# B&R Automation Studio project Teknologia25
Automation Studio 6.3.4.31; technology packages: mapp6D 3.4.1, mappView 6.3.2, OpcUaCs 6.0.0

## Configuration Config1

CPU X20EM0613, AutomationRuntime 6.0.2, Build 11.3.0, Vc 6.0.0

### Task classes (Cpu.sw)
```
Cyclic#1 (cycle 2000 us, tolerance 0 us):
  Main <- Main.Main.prg
  Acp6D <- Acp6D.Acp6D.prg
Cyclic#8:
  Robot <- Robot.Robot.prg
NcDataObjects: McDriveLog
Binaries: udbdef, mvLoader, mvConfig, OpcUaSrv, TCData, FWRules, ArSvcReg, BRRole, asfw, Role, ashwac, UaCsConfig, sysconf, iomap, Config_2, Config, Config_1, ashwd, User, arconfig
Libraries: operator, runtime, astime, AsIecCon, standard, RandLib, AsBrStr, AsBrMath, FileIO, BrAbbRws, AsHttp, ArEventLog, ArSsl, Crypto, AsIODiag, brdkMU, AsSem, sys_lib, brsystem, brdkSTR, MTFilter, MTTypes, MTLinAlg, AsUDP, AsTCP, comUtil, strUtil, McAcp6D, McBase, MpBase, brfiDemo
```

### Hardware
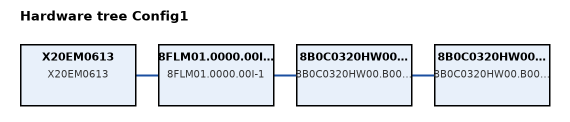
```
8B0C0320HW00.B00-1 : 8B0C0320HW00.B00-1 v1.0.1.3 (NodeNumber=3)  [PLK1 -> 8FLM01.0000.00I-1.PLK2 [Cable Type=PowerlinkCable, Length=10, Version=1.0.0.3]; PLK2 -> 8B0C0320HW00.B00-1_a.PLK1 [Cable Type=PowerlinkCable, Length=10, Version=1.0.0.3]]
  FunctionModel = DirectControl
  Supervision = off
  OutputVoltage = 58000
  CurrentLimitation = Used
  OutputCurrentLimit = 20000
  OutputCurrentLimitTime = 20
  ConfigOutputState = on
8B0C0320HW00.B00-1_a : 8B0C0320HW00.B00-1 v1.0.1.3  [PLK1 -> 8B0C0320HW00.B00-1.PLK2 [Cable Type=PowerlinkCable, Length=10, Version=1.0.0.3]]
  FunctionModel = DirectControl
  Supervision = off
  OutputVoltage = 58000
  CurrentLimitation = Used
  OutputCurrentLimit = 20000
  OutputCurrentLimitTime = 20
  ConfigOutputState = on
8FLM01.0000.00I-1 : 8FLM01.0000.00I-1 v1.0.0.1 (NodeNumber=239)  [PLK1 -> X20EM0613.IF3 [Cable Type=PowerlinkCable, Length=10, Version=1.0.0.3]; PLK2 -> 8B0C0320HW00.B00-1.PLK1 [Cable Type=PowerlinkCable, Length=10, Version=1.0.0.3]]
  Supervision = off
X20EM0613 : X20EM0613 v1.1.1.0
  Connector IF2:
    ActivateDevice = 1
    Mode = Manual
    InternetAddress = 192.168.125.201
    SubnetMask = 255.255.255.0
    ActivateSnmp = 2
  ConfigurationID = Teknologia25_Config1
  TimerDeviceType = EPLX2X
  TimerDevice = X20EM0613.IF3
  TaskClassIdleTime = 2000
  Cyclic1Duration = 2000
  Cyclic1Tolerance = 0
  FileDevice1
  FileDeviceName1 = 6DData
  FileDevicePath1 = USER_PATH
  ActivateFtpServer = 1
  FTPProtocol = 1
  FtpUser1
  FtpUsername1 = br
  FtpUserPassword1 = LZr6u6a2FqeMuMrXqkQdYPSQXL3utztiI9HOjYTJN4M=  // admin
  FtpUserSalt1 = xnOKDKah
  FTPAccessRight1 = 0
  FTPdevice1 = ALL
  ActivateWebServer = 1
  WebServerProtocol = 1
  WebServerPort = 8087
  ActivateSdm = 1
```

### IoMap.iom - X20EM0613/IoMap.iom
```iecst
VAR_CONFIG
	 Cyclic#1.::gCommInput.Array[0] AT %IW."8FLM01.0000.00I-1".EPL_FB_IN_0_I2007_S01;
	 Cyclic#1.::gCommInput.Array[1] AT %IW."8FLM01.0000.00I-1".EPL_FB_IN_1_I2007_S02;
	 Cyclic#1.::gCommInput.Array[2] AT %IW."8FLM01.0000.00I-1".EPL_FB_IN_2_I2007_S03;
	 Cyclic#1.::gCommInput.Array[3] AT %IW."8FLM01.0000.00I-1".EPL_FB_IN_3_I2007_S04;
	 Cyclic#1.::gCommInput.Array[4] AT %IW."8FLM01.0000.00I-1".EPL_FB_IN_4_I2007_S05;
	 Cyclic#1.::gCommInput.Array[5] AT %IW."8FLM01.0000.00I-1".EPL_FB_IN_5_I2007_S06;
	 Cyclic#1.::gCommInput.Array[6] AT %IW."8FLM01.0000.00I-1".EPL_FB_IN_6_I2007_S07;
	 Cyclic#1.::gCommInput.Array[7] AT %IW."8FLM01.0000.00I-1".EPL_FB_IN_7_I2007_S08;
	 Cyclic#1.::gCommInput.Array[8] AT %IW."8FLM01.0000.00I-1".EPL_FB_IN_8_I2007_S09;
	 Cyclic#1.::gCommInput.Array[9] AT %IW."8FLM01.0000.00I-1".EPL_FB_IN_9_I2007_S0A;
	 Cyclic#1.::gCommInput.Array[10] AT %IW."8FLM01.0000.00I-1".EPL_FB_IN_10_I2007_S0B;
	 Cyclic#1.::gCommInput.Array[11] AT %IW."8FLM01.0000.00I-1".EPL_FB_IN_11_I2007_S0C;
	 Cyclic#1.::gCommInput.Array[12] AT %IW."8FLM01.0000.00I-1".EPL_FB_IN_12_I2007_S0D;
	 Cyclic#1.::gCommInput.Array[13] AT %IW."8FLM01.0000.00I-1".EPL_FB_IN_13_I2007_S0E;
	 Cyclic#1.::gCommInput.Array[14] AT %IW."8FLM01.0000.00I-1".EPL_FB_IN_14_I2007_S0F;
	 Cyclic#1.::gCommInput.Array[15] AT %IW."8FLM01.0000.00I-1".EPL_FB_IN_15_I2007_S10;
	 Cyclic#1.::gCommInput.Array[16] AT %IW."8FLM01.0000.00I-1".EPL_FB_IN_16_I2007_S11;
	 Cyclic#1.::gCommInput.Array[17] AT %IW."8FLM01.0000.00I-1".EPL_FB_IN_17_I2007_S12;
	 Cyclic#1.::gCommInput.Array[18] AT %IW."8FLM01.0000.00I-1".EPL_FB_IN_18_I2007_S13;
	 Cyclic#1.::gCommInput.Array[19] AT %IW."8FLM01.0000.00I-1".EPL_FB_IN_19_I2007_S14;
	 Cyclic#1.::gCommInput.Array[20] AT %IW."8FLM01.0000.00I-1".EPL_FB_IN_20_I2007_S15;
	 Cyclic#1.::gCommInput.Array[21] AT %IW."8FLM01.0000.00I-1".EPL_FB_IN_21_I2007_S16;
	 Cyclic#1.::gCommInput.Array[22] AT %IW."8FLM01.0000.00I-1".EPL_FB_IN_22_I2007_S17;
	 Cyclic#1.::gCommInput.Array[23] AT %IW."8FLM01.0000.00I-1".EPL_FB_IN_23_I2007_S18;
	 Cyclic#1.::gCommInput.Array[24] AT %IW."8FLM01.0000.00I-1".EPL_FB_IN_24_I2007_S19;
	 Cyclic#1.::gCommInput.Array[25] AT %IW."8FLM01.0000.00I-1".EPL_FB_IN_25_I2007_S1A;
	 Cyclic#1.::gCommInput.Array[26] AT %IW."8FLM01.0000.00I-1".EPL_FB_IN_26_I2007_S1B;
	 Cyclic#1.::gCommInput.Array[27] AT %IW."8FLM01.0000.00I-1".EPL_FB_IN_27_I2007_S1C;
	 Cyclic#1.::gCommInput.Array[28] AT %IW."8FLM01.0000.00I-1".EPL_FB_IN_28_I2007_S1D;
	 Cyclic#1.::gCommInput.Array[29] AT %IW."8FLM01.0000.00I-1".EPL_FB_IN_29_I2007_S1E;
	 Cyclic#1.::gCommInput.Array[30] AT %IW."8FLM01.0000.00I-1".EPL_FB_IN_30_I2007_S1F;
	 Cyclic#1.::gCommInput.Array[31] AT %IW."8FLM01.0000.00I-1".EPL_FB_IN_31_I2007_S20;
	 Cyclic#1.::gCommInput.Array[32] AT %IW."8FLM01.0000.00I-1".EPL_FB_IN_32_I2007_S21;
	 Cyclic#1.::gCommInput.Array[33] AT %IW."8FLM01.0000.00I-1".EPL_FB_IN_33_I2007_S22;
	 Cyclic#1.::gCommInput.Array[34] AT %IW."8FLM01.0000.00I-1".EPL_FB_IN_34_I2007_S23;
	 Cyclic#1.::gCommInput.Array[35] AT %IW."8FLM01.0000.00I-1".EPL_FB_IN_35_I2007_S24;
	 Cyclic#1.::gCommInput.Array[36] AT %IW."8FLM01.0000.00I-1".EPL_FB_IN_36_I2007_S25;
	 Cyclic#1.::gCommInput.Array[37] AT %IW."8FLM01.0000.00I-1".EPL_FB_IN_37_I2007_S26;
	 Cyclic#1.::gCommInput.Array[38] AT %IW."8FLM01.0000.00I-1".EPL_FB_IN_38_I2007_S27;
	 Cyclic#1.::gCommInput.Array[39] AT %IW."8FLM01.0000.00I-1".EPL_FB_IN_39_I2007_S28;
	 Cyclic#1.::gCommInput.Array[40] AT %IW."8FLM01.0000.00I-1".EPL_FB_IN_40_I2007_S29;
	 Cyclic#1.::gCommInput.Array[41] AT %IW."8FLM01.0000.00I-1".EPL_FB_IN_41_I2007_S2A;
	 Cyclic#1.::gCommInput.Array[42] AT %IW."8FLM01.0000.00I-1".EPL_FB_IN_42_I2007_S2B;
	 Cyclic#1.::gCommInput.Array[43] AT %IW."8FLM01.0000.00I-1".EPL_FB_IN_43_I2007_S2C;
	 Cyclic#1.::gCommInput.Array[44] AT %IW."8FLM01.0000.00I-1".EPL_FB_IN_44_I2007_S2D;
	 Cyclic#1.::gCommInput.Array[45] AT %IW."8FLM01.0000.00I-1".EPL_FB_IN_45_I2007_S2E;
	 Cyclic#1.::gCommInput.Array[46] AT %IW."8FLM01.0000.00I-1".EPL_FB_IN_46_I2007_S2F;
	 Cyclic#1.::gCommInput.Array[47] AT %IW."8FLM01.0000.00I-1".EPL_FB_IN_47_I2007_S30;
	 Cyclic#1.::gCommInput.Array[48] AT %IW."8FLM01.0000.00I-1".EPL_FB_IN_48_I2007_S31;
	 Cyclic#1.::gCommInput.Array[49] AT %IW."8FLM01.0000.00I-1".EPL_FB_IN_49_I2007_S32;
	 Cyclic#1.::gCommInput.Array[50] AT %IW."8FLM01.0000.00I-1".EPL_FB_IN_50_I2007_S33;
	 Cyclic#1.::gCommInput.Array[51] AT %IW."8FLM01.0000.00I-1".EPL_FB_IN_51_I2007_S34;
	 Cyclic#1.::gCommInput.Array[52] AT %IW."8FLM01.0000.00I-1".EPL_FB_IN_52_I2007_S35;
	 Cyclic#1.::gCommInput.Array[53] AT %IW."8FLM01.0000.00I-1".EPL_FB_IN_53_I2007_S36;
	 Cyclic#1.::gCommInput.Array[54] AT %IW."8FLM01.0000.00I-1".EPL_FB_IN_54_I2007_S37;
	 Cyclic#1.::gCommInput.Array[55] AT %IW."8FLM01.0000.00I-1".EPL_FB_IN_55_I2007_S38;
	 Cyclic#1.::gCommInput.Array[56] AT %IW."8FLM01.0000.00I-1".EPL_FB_IN_56_I2007_S39;
	 Cyclic#1.::gCommInput.Array[57] AT %IW."8FLM01.0000.00I-1".EPL_FB_IN_57_I2007_S3A;
	 Cyclic#1.::gCommInput.Array[58] AT %IW."8FLM01.0000.00I-1".EPL_FB_IN_58_I2007_S3B;
	 Cyclic#1.::gCommInput.Array[59] AT %IW."8FLM01.0000.00I-1".EPL_FB_IN_59_I2007_S3C;
	 Cyclic#1.::gCommInput.Array[60] AT %IW."8FLM01.0000.00I-1".EPL_FB_IN_60_I2007_S3D;
	 Cyclic#1.::gCommInput.Array[61] AT %IW."8FLM01.0000.00I-1".EPL_FB_IN_61_I2007_S3E;
	 Cyclic#1.::gCommInput.Array[62] AT %IW."8FLM01.0000.00I-1".EPL_FB_IN_62_I2007_S3F;
	 Cyclic#1.::gCommInput.Array[63] AT %IW."8FLM01.0000.00I-1".EPL_FB_IN_63_I2007_S40;
	 Cyclic#1.::gCommInput.Array[64] AT %IW."8FLM01.0000.00I-1".EPL_FB_IN_64_I2007_S41;
	 Cyclic#1.::gCommInput.Array[65] AT %IW."8FLM01.0000.00I-1".EPL_FB_IN_65_I2007_S42;
	 Cyclic#1.::gCommInput.Array[66] AT %IW."8FLM01.0000.00I-1".EPL_FB_IN_66_I2007_S43;
	 Cyclic#1.::gCommInput.Array[67] AT %IW."8FLM01.0000.00I-1".EPL_FB_IN_67_I2007_S44;
	 Cyclic#1.::gCommInput.Array[68] AT %IW."8FLM01.0000.00I-1".EPL_FB_IN_68_I2007_S45;
	 Cyclic#1.::gCommInput.Array[69] AT %IW."8FLM01.0000.00I-1".EPL_FB_IN_69_I2007_S46;
	 Cyclic#1.::gCommInput.Array[70] AT %IW."8FLM01.0000.00I-1".EPL_FB_IN_70_I2007_S47;
	 Cyclic#1.::gCommInput.Array[71] AT %IW."8FLM01.0000.00I-1".EPL_FB_IN_71_I2007_S48;
	 Cyclic#1.::gCommInput.Array[72] AT %IW."8FLM01.0000.00I-1".EPL_FB_IN_72_I2007_S49;
	 Cyclic#1.::gCommInput.Array[73] AT %IW."8FLM01.0000.00I-1".EPL_FB_IN_73_I2007_S4A;
	 Cyclic#1.::gCommInput.Array[74] AT %IW."8FLM01.0000.00I-1".EPL_FB_IN_74_I2007_S4B;
	 Cyclic#1.::gCommInput.Array[75] AT %IW."8FLM01.0000.00I-1".EPL_FB_IN_75_I2007_S4C;
	 Cyclic#1.::gCommInput.Array[76] AT %IW."8FLM01.0000.00I-1".EPL_FB_IN_76_I2007_S4D;
	 Cyclic#1.::gCommInput.Array[77] AT %IW."8FLM01.0000.00I-1".EPL_FB_IN_77_I2007_S4E;
	 Cyclic#1.::gCommInput.Array[78] AT %IW."8FLM01.0000.00I-1".EPL_FB_IN_78_I2007_S4F;
	 Cyclic#1.::gCommInput.Array[79] AT %IW."8FLM01.0000.00I-1".EPL_FB_IN_79_I2007_S50;
	 Cyclic#1.::gCommInput.Array[80] AT %IW."8FLM01.0000.00I-1".EPL_FB_IN_80_I2007_S51;
	 Cyclic#1.::gCommInput.Array[81] AT %IW."8FLM01.0000.00I-1".EPL_FB_IN_81_I2007_S52;
	 Cyclic#1.::gCommInput.Array[82] AT %IW."8FLM01.0000.00I-1".EPL_FB_IN_82_I2007_S53;
	 Cyclic#1.::gCommInput.Array[83] AT %IW."8FLM01.0000.00I-1".EPL_FB_IN_83_I2007_S54;
	 Cyclic#1.::gCommInput.Array[84] AT %IW."8FLM01.0000.00I-1".EPL_FB_IN_84_I2007_S55;
	 Cyclic#1.::gCommInput.Array[85] AT %IW."8FLM01.0000.00I-1".EPL_FB_IN_85_I2007_S56;
	 Cyclic#1.::gCommInput.Array[86] AT %IW."8FLM01.0000.00I-1".EPL_FB_IN_86_I2007_S57;
	 Cyclic#1.::gCommInput.Array[87] AT %IW."8FLM01.0000.00I-1".EPL_FB_IN_87_I2007_S58;
	 Cyclic#1.::gCommInput.Array[88] AT %IW."8FLM01.0000.00I-1".EPL_FB_IN_88_I2007_S59;
	 Cyclic#1.::gCommInput.Array[89] AT %IW."8FLM01.0000.00I-1".EPL_FB_IN_89_I2007_S5A;
	 Cyclic#1.::gCommInput.Array[90] AT %IW."8FLM01.0000.00I-1".EPL_FB_IN_90_I2007_S5B;
	 Cyclic#1.::gCommInput.Array[91] AT %IW."8FLM01.0000.00I-1".EPL_FB_IN_91_I2007_S5C;
	 Cyclic#1.::gCommInput.Array[92] AT %IW."8FLM01.0000.00I-1".EPL_FB_IN_92_I2007_S5D;
	 Cyclic#1.::gCommInput.Array[93] AT %IW."8FLM01.0000.00I-1".EPL_FB_IN_93_I2007_S5E;
	 Cyclic#1.::gCommInput.Array[94] AT %IW."8FLM01.0000.00I-1".EPL_FB_IN_94_I2007_S5F;
	 Cyclic#1.::gCommInput.Array[95] AT %IW."8FLM01.0000.00I-1".EPL_FB_IN_95_I2007_S60;
	 Cyclic#1.::gCommInput.Array[96] AT %IW."8FLM01.0000.00I-1".EPL_FB_IN_96_I2007_S61;
	 Cyclic#1.::gCommInput.Array[97] AT %IW."8FLM01.0000.00I-1".EPL_FB_IN_97_I2007_S62;
	 Cyclic#1.::gCommInput.Array[98] AT %IW."8FLM01.0000.00I-1".EPL_FB_IN_98_I2007_S63;
	 Cyclic#1.::gCommInput.Array[99] AT %IW."8FLM01.0000.00I-1".EPL_FB_IN_99_I2007_S64;
	 Cyclic#1.::gCommInput.Array[100] AT %IW."8FLM01.0000.00I-1".EPL_FB_IN_100_I2007_S65;
	 Cyclic#1.::gCommInput.Array[101] AT %IW."8FLM01.0000.00I-1".EPL_FB_IN_101_I2007_S66;
	 Cyclic#1.::gCommInput.Array[102] AT %IW."8FLM01.0000.00I-1".EPL_FB_IN_102_I2007_S67;
	 Cyclic#1.::gCommInput.Array[103] AT %IW."8FLM01.0000.00I-1".EPL_FB_IN_103_I2007_S68;
	 Cyclic#1.::gCommInput.Array[104] AT %IW."8FLM01.0000.00I-1".EPL_FB_IN_104_I2007_S69;
	 Cyclic#1.::gCommInput.Array[105] AT %IW."8FLM01.0000.00I-1".EPL_FB_IN_105_I2007_S6A;
	 Cyclic#1.::gCommInput.Array[106] AT %IW."8FLM01.0000.00I-1".EPL_FB_IN_106_I2007_S6B;
	 Cyclic#1.::gCommInput.Array[107] AT %IW."8FLM01.0000.00I-1".EPL_FB_IN_107_I2007_S6C;
	 Cyclic#1.::gCommInput.Array[108] AT %IW."8FLM01.0000.00I-1".EPL_FB_IN_108_I2007_S6D;
	 Cyclic#1.::gCommInput.Array[109] AT %IW."8FLM01.0000.00I-1".EPL_FB_IN_109_I2007_S6E;
	 Cyclic#1.::gCommInput.Array[110] AT %IW."8FLM01.0000.00I-1".EPL_FB_IN_110_I2007_S6F;
	 Cyclic#1.::gCommInput.Array[111] AT %IW."8FLM01.0000.00I-1".EPL_FB_IN_111_I2007_S70;
	 Cyclic#1.::gCommInput.Array[112] AT %IW."8FLM01.0000.00I-1".EPL_FB_IN_112_I2007_S71;
	 Cyclic#1.::gCommInput.Array[113] AT %IW."8FLM01.0000.00I-1".EPL_FB_IN_113_I2007_S72;
	 Cyclic#1.::gCommInput.Array[114] AT %IW."8FLM01.0000.00I-1".EPL_FB_IN_114_I2007_S73;
	 Cyclic#1.::gCommInput.Array[115] AT %IW."8FLM01.0000.00I-1".EPL_FB_IN_115_I2007_S74;
	 Cyclic#1.::gCommInput.Array[116] AT %IW."8FLM01.0000.00I-1".EPL_FB_IN_116_I2007_S75;
	 Cyclic#1.::gCommInput.Array[117] AT %IW."8FLM01.0000.00I-1".EPL_FB_IN_117_I2007_S76;
	 Cyclic#1.::gCommInput.Array[118] AT %IW."8FLM01.0000.00I-1".EPL_FB_IN_118_I2007_S77;
	 Cyclic#1.::gCommInput.Array[119] AT %IW."8FLM01.0000.00I-1".EPL_FB_IN_119_I2007_S78;
	 Cyclic#1.::gCommInput.Array[120] AT %IW."8FLM01.0000.00I-1".EPL_FB_IN_120_I2007_S79;
	 Cyclic#1.::gCommInput.Array[121] AT %IW."8FLM01.0000.00I-1".EPL_FB_IN_121_I2007_S7A;
	 Cyclic#1.::gCommInput.Array[122] AT %IW."8FLM01.0000.00I-1".EPL_FB_IN_122_I2007_S7B;
	 Cyclic#1.::gCommInput.Array[123] AT %IW."8FLM01.0000.00I-1".EPL_FB_IN_123_I2007_S7C;
	 Cyclic#1.::gCommInput.Array[124] AT %IW."8FLM01.0000.00I-1".EPL_FB_IN_124_I2007_S7D;
	 Cyclic#1.::gCommInput.Array[125] AT %IW."8FLM01.0000.00I-1".EPL_FB_IN_125_I2007_S7E;
	 Cyclic#1.::gCommInput.Array[126] AT %IW."8FLM01.0000.00I-1".EPL_FB_IN_126_I2007_S7F;
	 Cyclic#1.::gCommInput.Array[127] AT %IW."8FLM01.0000.00I-1".EPL_FB_IN_127_I2007_S80;
	 Cyclic#1.::gCommInput.Array[128] AT %IW."8FLM01.0000.00I-1".EPL_FB_IN_128_I2007_S81;
	 Cyclic#1.::gCommInput.Array[129] AT %IW."8FLM01.0000.00I-1".EPL_FB_IN_129_I2007_S82;
	 Cyclic#1.::gCommInput.Array[130] AT %IW."8FLM01.0000.00I-1".EPL_FB_IN_130_I2007_S83;
	 Cyclic#1.::gCommInput.Array[131] AT %IW."8FLM01.0000.00I-1".EPL_FB_IN_131_I2007_S84;
	 Cyclic#1.::gCommInput.Array[132] AT %IW."8FLM01.0000.00I-1".EPL_FB_IN_132_I2007_S85;
	 Cyclic#1.::gCommInput.Array[133] AT %IW."8FLM01.0000.00I-1".EPL_FB_IN_133_I2007_S86;
	 Cyclic#1.::gCommInput.Array[134] AT %IW."8FLM01.0000.00I-1".EPL_FB_IN_134_I2007_S87;
	 Cyclic#1.::gCommInput.Array[135] AT %IW."8FLM01.0000.00I-1".EPL_FB_IN_135_I2007_S88;
	 Cyclic#1.::gCommInput.Array[136] AT %IW."8FLM01.0000.00I-1".EPL_FB_IN_136_I2007_S89;
	 Cyclic#1.::gCommInput.Array[137] AT %IW."8FLM01.0000.00I-1".EPL_FB_IN_137_I2007_S8A;
	 Cyclic#1.::gCommInput.Array[138] AT %IW."8FLM01.0000.00I-1".EPL_FB_IN_138_I2007_S8B;
	 Cyclic#1.::gCommInput.Array[139] AT %IW."8FLM01.0000.00I-1".EPL_FB_IN_139_I2007_S8C;
	 Cyclic#1.::gCommInput.Array[140] AT %IW."8FLM01.0000.00I-1".EPL_FB_IN_140_I2007_S8D;
	 Cyclic#1.::gCommInput.Array[141] AT %IW."8FLM01.0000.00I-1".EPL_FB_IN_141_I2007_S8E;
	 Cyclic#1.::gCommInput.Array[142] AT %IW."8FLM01.0000.00I-1".EPL_FB_IN_142_I2007_S8F;
	 Cyclic#1.::gCommInput.Array[143] AT %IW."8FLM01.0000.00I-1".EPL_FB_IN_143_I2007_S90;
	 Cyclic#1.::gCommInput.Array[144] AT %IW."8FLM01.0000.00I-1".EPL_FB_IN_144_I2007_S91;
	 Cyclic#1.::gCommInput.Array[145] AT %IW."8FLM01.0000.00I-1".EPL_FB_IN_145_I2007_S92;
	 Cyclic#1.::gCommInput.Array[146] AT %IW."8FLM01.0000.00I-1".EPL_FB_IN_146_I2007_S93;
	 Cyclic#1.::gCommInput.Array[147] AT %IW."8FLM01.0000.00I-1".EPL_FB_IN_147_I2007_S94;
	 Cyclic#1.::gCommInput.Array[148] AT %IW."8FLM01.0000.00I-1".EPL_FB_IN_148_I2007_S95;
	 Cyclic#1.::gCommInput.Array[149] AT %IW."8FLM01.0000.00I-1".EPL_FB_IN_149_I2007_S96;
	 Cyclic#1.::gCommInput.Array[150] AT %IW."8FLM01.0000.00I-1".EPL_FB_IN_150_I2007_S97;
	 Cyclic#1.::gCommInput.Array[151] AT %IW."8FLM01.0000.00I-1".EPL_FB_IN_151_I2007_S98;
	 Cyclic#1.::gCommInput.Array[152] AT %IW."8FLM01.0000.00I-1".EPL_FB_IN_152_I2007_S99;
	 Cyclic#1.::gCommInput.Array[153] AT %IW."8FLM01.0000.00I-1".EPL_FB_IN_153_I2007_S9A;
	 Cyclic#1.::gCommInput.Array[154] AT %IW."8FLM01.0000.00I-1".EPL_FB_IN_154_I2007_S9B;
	 Cyclic#1.::gCommInput.Array[155] AT %IW."8FLM01.0000.00I-1".EPL_FB_IN_155_I2007_S9C;
	 Cyclic#1.::gCommInput.Array[156] AT %IW."8FLM01.0000.00I-1".EPL_FB_IN_156_I2007_S9D;
	 Cyclic#1.::gCommInput.Array[157] AT %IW."8FLM01.0000.00I-1".EPL_FB_IN_157_I2007_S9E;
	 Cyclic#1.::gCommInput.Array[158] AT %IW."8FLM01.0000.00I-1".EPL_FB_IN_158_I2007_S9F;
	 Cyclic#1.::gCommInput.Array[159] AT %IW."8FLM01.0000.00I-1".EPL_FB_IN_159_I2007_SA0;
	 Cyclic#1.::gCommInput.Array[160] AT %IW."8FLM01.0000.00I-1".EPL_FB_IN_160_I2007_SA1;
	 Cyclic#1.::gCommInput.Array[161] AT %IW."8FLM01.0000.00I-1".EPL_FB_IN_161_I2007_SA2;
	 Cyclic#1.::gCommInput.Array[162] AT %IW."8FLM01.0000.00I-1".EPL_FB_IN_162_I2007_SA3;
	 Cyclic#1.::gCommInput.Array[163] AT %IW."8FLM01.0000.00I-1".EPL_FB_IN_163_I2007_SA4;
	 Cyclic#1.::gCommInput.Array[164] AT %IW."8FLM01.0000.00I-1".EPL_FB_IN_164_I2007_SA5;
	 Cyclic#1.::gCommInput.Array[165] AT %IW."8FLM01.0000.00I-1".EPL_FB_IN_165_I2007_SA6;
	 Cyclic#1.::gCommInput.Array[166] AT %IW."8FLM01.0000.00I-1".EPL_FB_IN_166_I2007_SA7;
	 Cyclic#1.::gCommInput.Array[167] AT %IW."8FLM01.0000.00I-1".EPL_FB_IN_167_I2007_SA8;
	 Cyclic#1.::gCommInput.Array[168] AT %IW."8FLM01.0000.00I-1".EPL_FB_IN_168_I2007_SA9;
	 Cyclic#1.::gCommInput.Array[169] AT %IW."8FLM01.0000.00I-1".EPL_FB_IN_169_I2007_SAA;
	 Cyclic#1.::gCommInput.Array[170] AT %IW."8FLM01.0000.00I-1".EPL_FB_IN_170_I2007_SAB;
	 Cyclic#1.::gCommInput.Array[171] AT %IW."8FLM01.0000.00I-1".EPL_FB_IN_171_I2007_SAC;
	 Cyclic#1.::gCommInput.Array[172] AT %IW."8FLM01.0000.00I-1".EPL_FB_IN_172_I2007_SAD;
	 Cyclic#1.::gCommInput.Array[173] AT %IW."8FLM01.0000.00I-1".EPL_FB_IN_173_I2007_SAE;
	 Cyclic#1.::gCommInput.Array[174] AT %IW."8FLM01.0000.00I-1".EPL_FB_IN_174_I2007_SAF;
	 Cyclic#1.::gCommInput.Array[175] AT %IW."8FLM01.0000.00I-1".EPL_FB_IN_175_I2007_SB0;
	 Cyclic#1.::gCommInput.Array[176] AT %IW."8FLM01.0000.00I-1".EPL_FB_IN_176_I2007_SB1;
	 Cyclic#1.::gCommInput.Array[177] AT %IW."8FLM01.0000.00I-1".EPL_FB_IN_177_I2007_SB2;
	 Cyclic#1.::gCommInput.Array[178] AT %IW."8FLM01.0000.00I-1".EPL_FB_IN_178_I2007_SB3;
	 Cyclic#1.::gCommInput.Array[179] AT %IW."8FLM01.0000.00I-1".EPL_FB_IN_179_I2007_SB4;
	 Cyclic#1.::gCommInput.Array[180] AT %IW."8FLM01.0000.00I-1".EPL_FB_IN_180_I2007_SB5;
	 Cyclic#1.::gCommInput.Array[181] AT %IW."8FLM01.0000.00I-1".EPL_FB_IN_181_I2007_SB6;
	 Cyclic#1.::gCommInput.Array[182] AT %IW."8FLM01.0000.00I-1".EPL_FB_IN_182_I2007_SB7;
	 Cyclic#1.::gCommInput.Array[183] AT %IW."8FLM01.0000.00I-1".EPL_FB_IN_183_I2007_SB8;
	 Cyclic#1.::gCommInput.Array[184] AT %IW."8FLM01.0000.00I-1".EPL_FB_IN_184_I2007_SB9;
	 Cyclic#1.::gCommInput.Array[185] AT %IW."8FLM01.0000.00I-1".EPL_FB_IN_185_I2007_SBA;
	 Cyclic#1.::gCommInput.Array[186] AT %IW."8FLM01.0000.00I-1".EPL_FB_IN_186_I2007_SBB;
	 Cyclic#1.::gCommInput.Array[187] AT %IW."8FLM01.0000.00I-1".EPL_FB_IN_187_I2007_SBC;
	 Cyclic#1.::gCommInput.Array[188] AT %IW."8FLM01.0000.00I-1".EPL_FB_IN_188_I2007_SBD;
	 Cyclic#1.::gCommInput.Array[189] AT %IW."8FLM01.0000.00I-1".EPL_FB_IN_189_I2007_SBE;
	 Cyclic#1.::gCommInput.Array[190] AT %IW."8FLM01.0000.00I-1".EPL_FB_IN_190_I2007_SBF;
	 Cyclic#1.::gCommInput.Array[191] AT %IW."8FLM01.0000.00I-1".EPL_FB_IN_191_I2007_SC0;
	 Cyclic#1.::gCommInput.Array[192] AT %IW."8FLM01.0000.00I-1".EPL_FB_IN_192_I2007_SC1;
	 Cyclic#1.::gCommInput.Array[193] AT %IW."8FLM01.0000.00I-1".EPL_FB_IN_193_I2007_SC2;
	 Cyclic#1.::gCommInput.Array[194] AT %IW."8FLM01.0000.00I-1".EPL_FB_IN_194_I2007_SC3;
	 Cyclic#1.::gCommInput.Array[195] AT %IW."8FLM01.0000.00I-1".EPL_FB_IN_195_I2007_SC4;
	 Cyclic#1.::gCommInput.Array[196] AT %IW."8FLM01.0000.00I-1".EPL_FB_IN_196_I2007_SC5;
	 Cyclic#1.::gCommInput.Array[197] AT %IW."8FLM01.0000.00I-1".EPL_FB_IN_197_I2007_SC6;
	 Cyclic#1.::gCommInput.Array[198] AT %IW."8FLM01.0000.00I-1".EPL_FB_IN_198_I2007_SC7;
	 Cyclic#1.::gCommInput.Array[199] AT %IW."8FLM01.0000.00I-1".EPL_FB_IN_199_I2007_SC8;
	 Cyclic#1.::gCommOutput.Array[0] AT %QW."8FLM01.0000.00I-1".EPL_FB_OUT_0_I2008_S01Out;
	 Cyclic#1.::gCommOutput.Array[1] AT %QW."8FLM01.0000.00I-1".EPL_FB_OUT_1_I2008_S02Out;
	 Cyclic#1.::gCommOutput.Array[2] AT %QW."8FLM01.0000.00I-1".EPL_FB_OUT_2_I2008_S03Out;
	 Cyclic#1.::gCommOutput.Array[3] AT %QW."8FLM01.0000.00I-1".EPL_FB_OUT_3_I2008_S04Out;
	 Cyclic#1.::gCommOutput.Array[4] AT %QW."8FLM01.0000.00I-1".EPL_FB_OUT_4_I2008_S05Out;
	 Cyclic#1.::gCommOutput.Array[5] AT %QW."8FLM01.0000.00I-1".EPL_FB_OUT_5_I2008_S06Out;
	 Cyclic#1.::gCommOutput.Array[6] AT %QW."8FLM01.0000.00I-1".EPL_FB_OUT_6_I2008_S07Out;
	 Cyclic#1.::gCommOutput.Array[7] AT %QW."8FLM01.0000.00I-1".EPL_FB_OUT_7_I2008_S08Out;
	 Cyclic#1.::gCommOutput.Array[8] AT %QW."8FLM01.0000.00I-1".EPL_FB_OUT_8_I2008_S09Out;
	 Cyclic#1.::gCommOutput.Array[9] AT %QW."8FLM01.0000.00I-1".EPL_FB_OUT_9_I2008_S0AOut;
	 Cyclic#1.::gCommOutput.Array[10] AT %QW."8FLM01.0000.00I-1".EPL_FB_OUT_10_I2008_S0BOut;
	 Cyclic#1.::gCommOutput.Array[11] AT %QW."8FLM01.0000.00I-1".EPL_FB_OUT_11_I2008_S0COut;
	 Cyclic#1.::gCommOutput.Array[12] AT %QW."8FLM01.0000.00I-1".EPL_FB_OUT_12_I2008_S0DOut;
	 Cyclic#1.::gCommOutput.Array[13] AT %QW."8FLM01.0000.00I-1".EPL_FB_OUT_13_I2008_S0EOut;
	 Cyclic#1.::gCommOutput.Array[14] AT %QW."8FLM01.0000.00I-1".EPL_FB_OUT_14_I2008_S0FOut;
	 Cyclic#1.::gCommOutput.Array[15] AT %QW."8FLM01.0000.00I-1".EPL_FB_OUT_15_I2008_S10Out;
	 Cyclic#1.::gCommOutput.Array[16] AT %QW."8FLM01.0000.00I-1".EPL_FB_OUT_16_I2008_S11Out;
	 Cyclic#1.::gCommOutput.Array[17] AT %QW."8FLM01.0000.00I-1".EPL_FB_OUT_17_I2008_S12Out;
	 Cyclic#1.::gCommOutput.Array[18] AT %QW."8FLM01.0000.00I-1".EPL_FB_OUT_18_I2008_S13Out;
	 Cyclic#1.::gCommOutput.Array[19] AT %QW."8FLM01.0000.00I-1".EPL_FB_OUT_19_I2008_S14Out;
	 Cyclic#1.::gCommOutput.Array[20] AT %QW."8FLM01.0000.00I-1".EPL_FB_OUT_20_I2008_S15Out;
	 Cyclic#1.::gCommOutput.Array[21] AT %QW."8FLM01.0000.00I-1".EPL_FB_OUT_21_I2008_S16Out;
	 Cyclic#1.::gCommOutput.Array[22] AT %QW."8FLM01.0000.00I-1".EPL_FB_OUT_22_I2008_S17Out;
	 Cyclic#1.::gCommOutput.Array[23] AT %QW."8FLM01.0000.00I-1".EPL_FB_OUT_23_I2008_S18Out;
	 Cyclic#1.::gCommOutput.Array[24] AT %QW."8FLM01.0000.00I-1".EPL_FB_OUT_24_I2008_S19Out;
	 Cyclic#1.::gCommOutput.Array[25] AT %QW."8FLM01.0000.00I-1".EPL_FB_OUT_25_I2008_S1AOut;
	 Cyclic#1.::gCommOutput.Array[26] AT %QW."8FLM01.0000.00I-1".EPL_FB_OUT_26_I2008_S1BOut;
	 Cyclic#1.::gCommOutput.Array[27] AT %QW."8FLM01.0000.00I-1".EPL_FB_OUT_27_I2008_S1COut;
	 Cyclic#1.::gCommOutput.Array[28] AT %QW."8FLM01.0000.00I-1".EPL_FB_OUT_28_I2008_S1DOut;
	 Cyclic#1.::gCommOutput.Array[29] AT %QW."8FLM01.0000.00I-1".EPL_FB_OUT_29_I2008_S1EOut;
	 Cyclic#1.::gCommOutput.Array[30] AT %QW."8FLM01.0000.00I-1".EPL_FB_OUT_30_I2008_S1FOut;
	 Cyclic#1.::gCommOutput.Array[31] AT %QW."8FLM01.0000.00I-1".EPL_FB_OUT_31_I2008_S20Out;
	 Cyclic#1.::gCommOutput.Array[32] AT %QW."8FLM01.0000.00I-1".EPL_FB_OUT_32_I2008_S21Out;
	 Cyclic#1.::gCommOutput.Array[33] AT %QW."8FLM01.0000.00I-1".EPL_FB_OUT_33_I2008_S22Out;
	 Cyclic#1.::gCommOutput.Array[34] AT %QW."8FLM01.0000.00I-1".EPL_FB_OUT_34_I2008_S23Out;
	 Cyclic#1.::gCommOutput.Array[35] AT %QW."8FLM01.0000.00I-1".EPL_FB_OUT_35_I2008_S24Out;
	 Cyclic#1.::gCommOutput.Array[36] AT %QW."8FLM01.0000.00I-1".EPL_FB_OUT_36_I2008_S25Out;
	 Cyclic#1.::gCommOutput.Array[37] AT %QW."8FLM01.0000.00I-1".EPL_FB_OUT_37_I2008_S26Out;
	 Cyclic#1.::gCommOutput.Array[38] AT %QW."8FLM01.0000.00I-1".EPL_FB_OUT_38_I2008_S27Out;
	 Cyclic#1.::gCommOutput.Array[39] AT %QW."8FLM01.0000.00I-1".EPL_FB_OUT_39_I2008_S28Out;
	 Cyclic#1.::gCommOutput.Array[40] AT %QW."8FLM01.0000.00I-1".EPL_FB_OUT_40_I2008_S29Out;
	 Cyclic#1.::gCommOutput.Array[41] AT %QW."8FLM01.0000.00I-1".EPL_FB_OUT_41_I2008_S2AOut;
	 Cyclic#1.::gCommOutput.Array[42] AT %QW."8FLM01.0000.00I-1".EPL_FB_OUT_42_I2008_S2BOut;
	 Cyclic#1.::gCommOutput.Array[43] AT %QW."8FLM01.0000.00I-1".EPL_FB_OUT_43_I2008_S2COut;
	 Cyclic#1.::gCommOutput.Array[44] AT %QW."8FLM01.0000.00I-1".EPL_FB_OUT_44_I2008_S2DOut;
	 Cyclic#1.::gCommOutput.Array[45] AT %QW."8FLM01.0000.00I-1".EPL_FB_OUT_45_I2008_S2EOut;
	 Cyclic#1.::gCommOutput.Array[46] AT %QW."8FLM01.0000.00I-1".EPL_FB_OUT_46_I2008_S2FOut;
	 Cyclic#1.::gCommOutput.Array[47] AT %QW."8FLM01.0000.00I-1".EPL_FB_OUT_47_I2008_S30Out;
	 Cyclic#1.::gCommOutput.Array[48] AT %QW."8FLM01.0000.00I-1".EPL_FB_OUT_48_I2008_S31Out;
	 Cyclic#1.::gCommOutput.Array[49] AT %QW."8FLM01.0000.00I-1".EPL_FB_OUT_49_I2008_S32Out;
	 Cyclic#1.::gCommOutput.Array[50] AT %QW."8FLM01.0000.00I-1".EPL_FB_OUT_50_I2008_S33Out;
	 Cyclic#1.::gCommOutput.Array[51] AT %QW."8FLM01.0000.00I-1".EPL_FB_OUT_51_I2008_S34Out;
	 Cyclic#1.::gCommOutput.Array[52] AT %QW."8FLM01.0000.00I-1".EPL_FB_OUT_52_I2008_S35Out;
	 Cyclic#1.::gCommOutput.Array[53] AT %QW."8FLM01.0000.00I-1".EPL_FB_OUT_53_I2008_S36Out;
	 Cyclic#1.::gCommOutput.Array[54] AT %QW."8FLM01.0000.00I-1".EPL_FB_OUT_54_I2008_S37Out;
	 Cyclic#1.::gCommOutput.Array[55] AT %QW."8FLM01.0000.00I-1".EPL_FB_OUT_55_I2008_S38Out;
	 Cyclic#1.::gCommOutput.Array[56] AT %QW."8FLM01.0000.00I-1".EPL_FB_OUT_56_I2008_S39Out;
	 Cyclic#1.::gCommOutput.Array[57] AT %QW."8FLM01.0000.00I-1".EPL_FB_OUT_57_I2008_S3AOut;
	 Cyclic#1.::gCommOutput.Array[58] AT %QW."8FLM01.0000.00I-1".EPL_FB_OUT_58_I2008_S3BOut;
	 Cyclic#1.::gCommOutput.Array[59] AT %QW."8FLM01.0000.00I-1".EPL_FB_OUT_59_I2008_S3COut;
	 Cyclic#1.::gCommOutput.Array[60] AT %QW."8FLM01.0000.00I-1".EPL_FB_OUT_60_I2008_S3DOut;
	 Cyclic#1.::gCommOutput.Array[61] AT %QW."8FLM01.0000.00I-1".EPL_FB_OUT_61_I2008_S3EOut;
	 Cyclic#1.::gCommOutput.Array[62] AT %QW."8FLM01.0000.00I-1".EPL_FB_OUT_62_I2008_S3FOut;
	 Cyclic#1.::gCommOutput.Array[63] AT %QW."8FLM01.0000.00I-1".EPL_FB_OUT_63_I2008_S40Out;
	 Cyclic#1.::gCommOutput.Array[64] AT %QW."8FLM01.0000.00I-1".EPL_FB_OUT_64_I2008_S41Out;
	 Cyclic#1.::gCommOutput.Array[65] AT %QW."8FLM01.0000.00I-1".EPL_FB_OUT_65_I2008_S42Out;
	 Cyclic#1.::gCommOutput.Array[66] AT %QW."8FLM01.0000.00I-1".EPL_FB_OUT_66_I2008_S43Out;
	 Cyclic#1.::gCommOutput.Array[67] AT %QW."8FLM01.0000.00I-1".EPL_FB_OUT_67_I2008_S44Out;
	 Cyclic#1.::gCommOutput.Array[68] AT %QW."8FLM01.0000.00I-1".EPL_FB_OUT_68_I2008_S45Out;
	 Cyclic#1.::gCommOutput.Array[69] AT %QW."8FLM01.0000.00I-1".EPL_FB_OUT_69_I2008_S46Out;
	 Cyclic#1.::gCommOutput.Array[70] AT %QW."8FLM01.0000.00I-1".EPL_FB_OUT_70_I2008_S47Out;
	 Cyclic#1.::gCommOutput.Array[71] AT %QW."8FLM01.0000.00I-1".EPL_FB_OUT_71_I2008_S48Out;
	 Cyclic#1.::gCommOutput.Array[72] AT %QW."8FLM01.0000.00I-1".EPL_FB_OUT_72_I2008_S49Out;
	 Cyclic#1.::gCommOutput.Array[73] AT %QW."8FLM01.0000.00I-1".EPL_FB_OUT_73_I2008_S4AOut;
	 Cyclic#1.::gCommOutput.Array[74] AT %QW."8FLM01.0000.00I-1".EPL_FB_OUT_74_I2008_S4BOut;
	 Cyclic#1.::gCommOutput.Array[75] AT %QW."8FLM01.0000.00I-1".EPL_FB_OUT_75_I2008_S4COut;
	 Cyclic#1.::gCommOutput.Array[76] AT %QW."8FLM01.0000.00I-1".EPL_FB_OUT_76_I2008_S4DOut;
	 Cyclic#1.::gCommOutput.Array[77] AT %QW."8FLM01.0000.00I-1".EPL_FB_OUT_77_I2008_S4EOut;
	 Cyclic#1.::gCommOutput.Array[78] AT %QW."8FLM01.0000.00I-1".EPL_FB_OUT_78_I2008_S4FOut;
	 Cyclic#1.::gCommOutput.Array[79] AT %QW."8FLM01.0000.00I-1".EPL_FB_OUT_79_I2008_S50Out;
	 Cyclic#1.::gCommOutput.Array[80] AT %QW."8FLM01.0000.00I-1".EPL_FB_OUT_80_I2008_S51Out;
	 Cyclic#1.::gCommOutput.Array[81] AT %QW."8FLM01.0000.00I-1".EPL_FB_OUT_81_I2008_S52Out;
	 Cyclic#1.::gCommOutput.Array[82] AT %QW."8FLM01.0000.00I-1".EPL_FB_OUT_82_I2008_S53Out;
	 Cyclic#1.::gCommOutput.Array[83] AT %QW."8FLM01.0000.00I-1".EPL_FB_OUT_83_I2008_S54Out;
	 Cyclic#1.::gCommOutput.Array[84] AT %QW."8FLM01.0000.00I-1".EPL_FB_OUT_84_I2008_S55Out;
	 Cyclic#1.::gCommOutput.Array[85] AT %QW."8FLM01.0000.00I-1".EPL_FB_OUT_85_I2008_S56Out;
	 Cyclic#1.::gCommOutput.Array[86] AT %QW."8FLM01.0000.00I-1".EPL_FB_OUT_86_I2008_S57Out;
	 Cyclic#1.::gCommOutput.Array[87] AT %QW."8FLM01.0000.00I-1".EPL_FB_OUT_87_I2008_S58Out;
	 Cyclic#1.::gCommOutput.Array[88] AT %QW."8FLM01.0000.00I-1".EPL_FB_OUT_88_I2008_S59Out;
	 Cyclic#1.::gCommOutput.Array[89] AT %QW."8FLM01.0000.00I-1".EPL_FB_OUT_89_I2008_S5AOut;
	 Cyclic#1.::gCommOutput.Array[90] AT %QW."8FLM01.0000.00I-1".EPL_FB_OUT_90_I2008_S5BOut;
	 Cyclic#1.::gCommOutput.Array[91] AT %QW."8FLM01.0000.00I-1".EPL_FB_OUT_91_I2008_S5COut;
	 Cyclic#1.::gCommOutput.Array[92] AT %QW."8FLM01.0000.00I-1".EPL_FB_OUT_92_I2008_S5DOut;
	 Cyclic#1.::gCommOutput.Array[93] AT %QW."8FLM01.0000.00I-1".EPL_FB_OUT_93_I2008_S5EOut;
	 Cyclic#1.::gCommOutput.Array[94] AT %QW."8FLM01.0000.00I-1".EPL_FB_OUT_94_I2008_S5FOut;
	 Cyclic#1.::gCommOutput.Array[95] AT %QW."8FLM01.0000.00I-1".EPL_FB_OUT_95_I2008_S60Out;
	 Cyclic#1.::gCommOutput.Array[96] AT %QW."8FLM01.0000.00I-1".EPL_FB_OUT_96_I2008_S61Out;
	 Cyclic#1.::gCommOutput.Array[97] AT %QW."8FLM01.0000.00I-1".EPL_FB_OUT_97_I2008_S62Out;
	 Cyclic#1.::gCommOutput.Array[98] AT %QW."8FLM01.0000.00I-1".EPL_FB_OUT_98_I2008_S63Out;
	 Cyclic#1.::gCommOutput.Array[99] AT %QW."8FLM01.0000.00I-1".EPL_FB_OUT_99_I2008_S64Out;
	 Cyclic#1.::gCommOutput.Array[100] AT %QW."8FLM01.0000.00I-1".EPL_FB_OUT_100_I2008_S65Out;
	 Cyclic#1.::gCommOutput.Array[101] AT %QW."8FLM01.0000.00I-1".EPL_FB_OUT_101_I2008_S66Out;
	 Cyclic#1.::gCommOutput.Array[102] AT %QW."8FLM01.0000.00I-1".EPL_FB_OUT_102_I2008_S67Out;
	 Cyclic#1.::gCommOutput.Array[103] AT %QW."8FLM01.0000.00I-1".EPL_FB_OUT_103_I2008_S68Out;
	 Cyclic#1.::gCommOutput.Array[104] AT %QW."8FLM01.0000.00I-1".EPL_FB_OUT_104_I2008_S69Out;
	 Cyclic#1.::gCommOutput.Array[105] AT %QW."8FLM01.0000.00I-1".EPL_FB_OUT_105_I2008_S6AOut;
	 Cyclic#1.::gCommOutput.Array[106] AT %QW."8FLM01.0000.00I-1".EPL_FB_OUT_106_I2008_S6BOut;
	 Cyclic#1.::gCommOutput.Array[107] AT %QW."8FLM01.0000.00I-1".EPL_FB_OUT_107_I2008_S6COut;
	 Cyclic#1.::gCommOutput.Array[108] AT %QW."8FLM01.0000.00I-1".EPL_FB_OUT_108_I2008_S6DOut;
	 Cyclic#1.::gCommOutput.Array[109] AT %QW."8FLM01.0000.00I-1".EPL_FB_OUT_109_I2008_S6EOut;
	 Cyclic#1.::gCommOutput.Array[110] AT %QW."8FLM01.0000.00I-1".EPL_FB_OUT_110_I2008_S6FOut;
	 Cyclic#1.::gCommOutput.Array[111] AT %QW."8FLM01.0000.00I-1".EPL_FB_OUT_111_I2008_S70Out;
	 Cyclic#1.::gCommOutput.Array[112] AT %QW."8FLM01.0000.00I-1".EPL_FB_OUT_112_I2008_S71Out;
	 Cyclic#1.::gCommOutput.Array[113] AT %QW."8FLM01.0000.00I-1".EPL_FB_OUT_113_I2008_S72Out;
	 Cyclic#1.::gCommOutput.Array[114] AT %QW."8FLM01.0000.00I-1".EPL_FB_OUT_114_I2008_S73Out;
	 Cyclic#1.::gCommOutput.Array[115] AT %QW."8FLM01.0000.00I-1".EPL_FB_OUT_115_I2008_S74Out;
	 Cyclic#1.::gCommOutput.Array[116] AT %QW."8FLM01.0000.00I-1".EPL_FB_OUT_116_I2008_S75Out;
	 Cyclic#1.::gCommOutput.Array[117] AT %QW."8FLM01.0000.00I-1".EPL_FB_OUT_117_I2008_S76Out;
	 Cyclic#1.::gCommOutput.Array[118] AT %QW."8FLM01.0000.00I-1".EPL_FB_OUT_118_I2008_S77Out;
	 Cyclic#1.::gCommOutput.Array[119] AT %QW."8FLM01.0000.00I-1".EPL_FB_OUT_119_I2008_S78Out;
	 Cyclic#1.::gCommOutput.Array[120] AT %QW."8FLM01.0000.00I-1".EPL_FB_OUT_120_I2008_S79Out;
	 Cyclic#1.::gCommOutput.Array[121] AT %QW."8FLM01.0000.00I-1".EPL_FB_OUT_121_I2008_S7AOut;
	 Cyclic#1.::gCommOutput.Array[122] AT %QW."8FLM01.0000.00I-1".EPL_FB_OUT_122_I2008_S7BOut;
	 Cyclic#1.::gCommOutput.Array[123] AT %QW."8FLM01.0000.00I-1".EPL_FB_OUT_123_I2008_S7COut;
	 Cyclic#1.::gCommOutput.Array[124] AT %QW."8FLM01.0000.00I-1".EPL_FB_OUT_124_I2008_S7DOut;
	 Cyclic#1.::gCommOutput.Array[125] AT %QW."8FLM01.0000.00I-1".EPL_FB_OUT_125_I2008_S7EOut;
	 Cyclic#1.::gCommOutput.Array[126] AT %QW."8FLM01.0000.00I-1".EPL_FB_OUT_126_I2008_S7FOut;
	 Cyclic#1.::gCommOutput.Array[127] AT %QW."8FLM01.0000.00I-1".EPL_FB_OUT_127_I2008_S80Out;
	 Cyclic#1.::gCommOutput.Array[128] AT %QW."8FLM01.0000.00I-1".EPL_FB_OUT_128_I2008_S81Out;
	 Cyclic#1.::gCommOutput.Array[129] AT %QW."8FLM01.0000.00I-1".EPL_FB_OUT_129_I2008_S82Out;
	 Cyclic#1.::gCommOutput.Array[130] AT %QW."8FLM01.0000.00I-1".EPL_FB_OUT_130_I2008_S83Out;
	 Cyclic#1.::gCommOutput.Array[131] AT %QW."8FLM01.0000.00I-1".EPL_FB_OUT_131_I2008_S84Out;
	 Cyclic#1.::gCommOutput.Array[132] AT %QW."8FLM01.0000.00I-1".EPL_FB_OUT_132_I2008_S85Out;
	 Cyclic#1.::gCommOutput.Array[133] AT %QW."8FLM01.0000.00I-1".EPL_FB_OUT_133_I2008_S86Out;
	 Cyclic#1.::gCommOutput.Array[134] AT %QW."8FLM01.0000.00I-1".EPL_FB_OUT_134_I2008_S87Out;
	 Cyclic#1.::gCommOutput.Array[135] AT %QW."8FLM01.0000.00I-1".EPL_FB_OUT_135_I2008_S88Out;
	 Cyclic#1.::gCommOutput.Array[136] AT %QW."8FLM01.0000.00I-1".EPL_FB_OUT_136_I2008_S89Out;
	 Cyclic#1.::gCommOutput.Array[137] AT %QW."8FLM01.0000.00I-1".EPL_FB_OUT_137_I2008_S8AOut;
	 Cyclic#1.::gCommOutput.Array[138] AT %QW."8FLM01.0000.00I-1".EPL_FB_OUT_138_I2008_S8BOut;
	 Cyclic#1.::gCommOutput.Array[139] AT %QW."8FLM01.0000.00I-1".EPL_FB_OUT_139_I2008_S8COut;
	 Cyclic#1.::gCommOutput.Array[140] AT %QW."8FLM01.0000.00I-1".EPL_FB_OUT_140_I2008_S8DOut;
	 Cyclic#1.::gCommOutput.Array[141] AT %QW."8FLM01.0000.00I-1".EPL_FB_OUT_141_I2008_S8EOut;
	 Cyclic#1.::gCommOutput.Array[142] AT %QW."8FLM01.0000.00I-1".EPL_FB_OUT_142_I2008_S8FOut;
	 Cyclic#1.::gCommOutput.Array[143] AT %QW."8FLM01.0000.00I-1".EPL_FB_OUT_143_I2008_S90Out;
	 Cyclic#1.::gCommOutput.Array[144] AT %QW."8FLM01.0000.00I-1".EPL_FB_OUT_144_I2008_S91Out;
	 Cyclic#1.::gCommOutput.Array[145] AT %QW."8FLM01.0000.00I-1".EPL_FB_OUT_145_I2008_S92Out;
	 Cyclic#1.::gCommOutput.Array[146] AT %QW."8FLM01.0000.00I-1".EPL_FB_OUT_146_I2008_S93Out;
	 Cyclic#1.::gCommOutput.Array[147] AT %QW."8FLM01.0000.00I-1".EPL_FB_OUT_147_I2008_S94Out;
	 Cyclic#1.::gCommOutput.Array[148] AT %QW."8FLM01.0000.00I-1".EPL_FB_OUT_148_I2008_S95Out;
	 Cyclic#1.::gCommOutput.Array[149] AT %QW."8FLM01.0000.00I-1".EPL_FB_OUT_149_I2008_S96Out;
	 Cyclic#1.::gCommOutput.Array[150] AT %QW."8FLM01.0000.00I-1".EPL_FB_OUT_150_I2008_S97Out;
	 Cyclic#1.::gCommOutput.Array[151] AT %QW."8FLM01.0000.00I-1".EPL_FB_OUT_151_I2008_S98Out;
	 Cyclic#1.::gCommOutput.Array[152] AT %QW."8FLM01.0000.00I-1".EPL_FB_OUT_152_I2008_S99Out;
	 Cyclic#1.::gCommOutput.Array[153] AT %QW."8FLM01.0000.00I-1".EPL_FB_OUT_153_I2008_S9AOut;
	 Cyclic#1.::gCommOutput.Array[154] AT %QW."8FLM01.0000.00I-1".EPL_FB_OUT_154_I2008_S9BOut;
	 Cyclic#1.::gCommOutput.Array[155] AT %QW."8FLM01.0000.00I-1".EPL_FB_OUT_155_I2008_S9COut;
	 Cyclic#1.::gCommOutput.Array[156] AT %QW."8FLM01.0000.00I-1".EPL_FB_OUT_156_I2008_S9DOut;
	 Cyclic#1.::gCommOutput.Array[157] AT %QW."8FLM01.0000.00I-1".EPL_FB_OUT_157_I2008_S9EOut;
	 Cyclic#1.::gCommOutput.Array[158] AT %QW."8FLM01.0000.00I-1".EPL_FB_OUT_158_I2008_S9FOut;
	 Cyclic#1.::gCommOutput.Array[159] AT %QW."8FLM01.0000.00I-1".EPL_FB_OUT_159_I2008_SA0Out;
	 Cyclic#1.::gCommOutput.Array[160] AT %QW."8FLM01.0000.00I-1".EPL_FB_OUT_160_I2008_SA1Out;
	 Cyclic#1.::gCommOutput.Array[161] AT %QW."8FLM01.0000.00I-1".EPL_FB_OUT_161_I2008_SA2Out;
	 Cyclic#1.::gCommOutput.Array[162] AT %QW."8FLM01.0000.00I-1".EPL_FB_OUT_162_I2008_SA3Out;
	 Cyclic#1.::gCommOutput.Array[163] AT %QW."8FLM01.0000.00I-1".EPL_FB_OUT_163_I2008_SA4Out;
	 Cyclic#1.::gCommOutput.Array[164] AT %QW."8FLM01.0000.00I-1".EPL_FB_OUT_164_I2008_SA5Out;
	 Cyclic#1.::gCommOutput.Array[165] AT %QW."8FLM01.0000.00I-1".EPL_FB_OUT_165_I2008_SA6Out;
	 Cyclic#1.::gCommOutput.Array[166] AT %QW."8FLM01.0000.00I-1".EPL_FB_OUT_166_I2008_SA7Out;
	 Cyclic#1.::gCommOutput.Array[167] AT %QW."8FLM01.0000.00I-1".EPL_FB_OUT_167_I2008_SA8Out;
	 Cyclic#1.::gCommOutput.Array[168] AT %QW."8FLM01.0000.00I-1".EPL_FB_OUT_168_I2008_SA9Out;
	 Cyclic#1.::gCommOutput.Array[169] AT %QW."8FLM01.0000.00I-1".EPL_FB_OUT_169_I2008_SAAOut;
	 Cyclic#1.::gCommOutput.Array[170] AT %QW."8FLM01.0000.00I-1".EPL_FB_OUT_170_I2008_SABOut;
	 Cyclic#1.::gCommOutput.Array[171] AT %QW."8FLM01.0000.00I-1".EPL_FB_OUT_171_I2008_SACOut;
	 Cyclic#1.::gCommOutput.Array[172] AT %QW."8FLM01.0000.00I-1".EPL_FB_OUT_172_I2008_SADOut;
	 Cyclic#1.::gCommOutput.Array[173] AT %QW."8FLM01.0000.00I-1".EPL_FB_OUT_173_I2008_SAEOut;
	 Cyclic#1.::gCommOutput.Array[174] AT %QW."8FLM01.0000.00I-1".EPL_FB_OUT_174_I2008_SAFOut;
	 Cyclic#1.::gCommOutput.Array[175] AT %QW."8FLM01.0000.00I-1".EPL_FB_OUT_175_I2008_SB0Out;
	 Cyclic#1.::gCommOutput.Array[176] AT %QW."8FLM01.0000.00I-1".EPL_FB_OUT_176_I2008_SB1Out;
	 Cyclic#1.::gCommOutput.Array[177] AT %QW."8FLM01.0000.00I-1".EPL_FB_OUT_177_I2008_SB2Out;
	 Cyclic#1.::gCommOutput.Array[178] AT %QW."8FLM01.0000.00I-1".EPL_FB_OUT_178_I2008_SB3Out;
	 Cyclic#1.::gCommOutput.Array[179] AT %QW."8FLM01.0000.00I-1".EPL_FB_OUT_179_I2008_SB4Out;
	 Cyclic#1.::gCommOutput.Array[180] AT %QW."8FLM01.0000.00I-1".EPL_FB_OUT_180_I2008_SB5Out;
	 Cyclic#1.::gCommOutput.Array[181] AT %QW."8FLM01.0000.00I-1".EPL_FB_OUT_181_I2008_SB6Out;
	 Cyclic#1.::gCommOutput.Array[182] AT %QW."8FLM01.0000.00I-1".EPL_FB_OUT_182_I2008_SB7Out;
	 Cyclic#1.::gCommOutput.Array[183] AT %QW."8FLM01.0000.00I-1".EPL_FB_OUT_183_I2008_SB8Out;
	 Cyclic#1.::gCommOutput.Array[184] AT %QW."8FLM01.0000.00I-1".EPL_FB_OUT_184_I2008_SB9Out;
	 Cyclic#1.::gCommOutput.Array[185] AT %QW."8FLM01.0000.00I-1".EPL_FB_OUT_185_I2008_SBAOut;
	 Cyclic#1.::gCommOutput.Array[186] AT %QW."8FLM01.0000.00I-1".EPL_FB_OUT_186_I2008_SBBOut;
	 Cyclic#1.::gCommOutput.Array[187] AT %QW."8FLM01.0000.00I-1".EPL_FB_OUT_187_I2008_SBCOut;
	 Cyclic#1.::gCommOutput.Array[188] AT %QW."8FLM01.0000.00I-1".EPL_FB_OUT_188_I2008_SBDOut;
	 Cyclic#1.::gCommOutput.Array[189] AT %QW."8FLM01.0000.00I-1".EPL_FB_OUT_189_I2008_SBEOut;
	 Cyclic#1.::gCommOutput.Array[190] AT %QW."8FLM01.0000.00I-1".EPL_FB_OUT_190_I2008_SBFOut;
	 Cyclic#1.::gCommOutput.Array[191] AT %QW."8FLM01.0000.00I-1".EPL_FB_OUT_191_I2008_SC0Out;
	 Cyclic#1.::gCommOutput.Array[192] AT %QW."8FLM01.0000.00I-1".EPL_FB_OUT_192_I2008_SC1Out;
	 Cyclic#1.::gCommOutput.Array[193] AT %QW."8FLM01.0000.00I-1".EPL_FB_OUT_193_I2008_SC2Out;
	 Cyclic#1.::gCommOutput.Array[194] AT %QW."8FLM01.0000.00I-1".EPL_FB_OUT_194_I2008_SC3Out;
	 Cyclic#1.::gCommOutput.Array[195] AT %QW."8FLM01.0000.00I-1".EPL_FB_OUT_195_I2008_SC4Out;
	 Cyclic#1.::gCommOutput.Array[196] AT %QW."8FLM01.0000.00I-1".EPL_FB_OUT_196_I2008_SC5Out;
	 Cyclic#1.::gCommOutput.Array[197] AT %QW."8FLM01.0000.00I-1".EPL_FB_OUT_197_I2008_SC6Out;
	 Cyclic#1.::gCommOutput.Array[198] AT %QW."8FLM01.0000.00I-1".EPL_FB_OUT_198_I2008_SC7Out;
	 Cyclic#1.::gCommOutput.Array[199] AT %QW."8FLM01.0000.00I-1".EPL_FB_OUT_199_I2008_SC8Out;
END_VAR
```

### Config_1.layout6d - X20EM0613/mapp6D/Config_1.layout6d
```
Element Layout6D_1 (Type=layout6d)
  GridSize = 0
  UserOrigin:
    OffsetX = 0
    OffsetY = 0
  Segments:
    SegRow = 4
    SegCol = 4
    Segment[1]:
      TypeGrid240 = 0
      TypeGrid120 = 0
      TypeGrid320 = 0
      TypeGrid160 = 0
      X = 0
      Y = 0
      Name
      IsMaster = True
      PowerSectorName
      Gaps:
        Left = 0
        Bottom = 0
        Right = 0
        Top = 0
        S4Left = 0
        S4Bottom = 0
        S4Right = 0
        S4Top = 0
      BorderID:
        Left = 0
        Bottom = 0
        Right = 0
        Top = 0
    Segment[2]:
      TypeGrid240 = 0
      TypeGrid120 = 0
      TypeGrid320 = 0
      TypeGrid160 = 0
      X = 0
      Y = 1
      Name
      IsMaster = False
      PowerSectorName
      Gaps:
        Left = 0
        Bottom = 0
        Right = 0
        Top = 0
        S4Left = 0
        S4Bottom = 0
        S4Right = 0
        S4Top = 0
      BorderID:
        Left = 0
        Bottom = 0
        Right = 0
        Top = 0
    Segment[3]:
      TypeGrid240 = 0
      TypeGrid120 = 0
      TypeGrid320 = 0
      TypeGrid160 = 0
      X = 0
      Y = 2
      Name
      IsMaster = False
      PowerSectorName
      Gaps:
        Left = 0
        Bottom = 0
        Right = 0
        Top = 0
        S4Left = 0
        S4Bottom = 0
        S4Right = 0
        S4Top = 0
      BorderID:
        Left = 0
        Bottom = 0
        Right = 0
        Top = 0
    Segment[4]:
      TypeGrid240 = 0
      TypeGrid120 = 0
      TypeGrid320 = 0
      TypeGrid160 = 0
      X = 0
      Y = 3
      Name
      IsMaster = False
      PowerSectorName
      Gaps:
        Left = 0
        Bottom = 0
        Right = 0
        Top = 0
        S4Left = 0
        S4Bottom = 0
        S4Right = 0
        S4Top = 0
      BorderID:
        Left = 0
        Bottom = 0
        Right = 0
        Top = 0
    Segment[5]:
      TypeGrid240 = 0
      TypeGrid120 = 0
      TypeGrid320 = 0
      TypeGrid160 = 0
      X = 1
      Y = 0
      Name
      IsMaster = False
      PowerSectorName
      Gaps:
        Left = 0
        Bottom = 0
        Right = 0
        Top = 0
        S4Left = 0
        S4Bottom = 0
        S4Right = 0
        S4Top = 0
      BorderID:
        Left = 0
        Bottom = 0
        Right = 0
        Top = 0
    Segment[6]:
      TypeGrid240 = 0
      TypeGrid120 = 0
      TypeGrid320 = 0
      TypeGrid160 = 0
      X = 1
      Y = 1
      Name
      IsMaster = False
      PowerSectorName
      Gaps:
        Left = 0
        Bottom = 0
        Right = 0
        Top = 0
        S4Left = 0
        S4Bottom = 0
        S4Right = 0
        S4Top = 0
      BorderID:
        Left = 0
        Bottom = 0
        Right = 0
        Top = 0
    Segment[7]:
      TypeGrid240 = 0
      TypeGrid120 = 0
      TypeGrid320 = 0
      TypeGrid160 = 0
      X = 1
      Y = 2
      Name
      IsMaster = False
      PowerSectorName
      Gaps:
        Left = 0
        Bottom = 0
        Right = 0
        Top = 0
        S4Left = 0
        S4Bottom = 0
        S4Right = 0
        S4Top = 0
      BorderID:
        Left = 0
        Bottom = 0
        Right = 0
        Top = 0
    Segment[8]:
      TypeGrid240 = 0
      TypeGrid120 = 0
      TypeGrid320 = 0
      TypeGrid160 = 0
      X = 1
      Y = 3
      Name
      IsMaster = False
      PowerSectorName
      Gaps:
        Left = 0
        Bottom = 0
        Right = 0
        Top = 0
        S4Left = 0
        S4Bottom = 0
        S4Right = 0
        S4Top = 0
      BorderID:
        Left = 0
        Bottom = 0
        Right = 0
        Top = 0
    Segment[9]:
      TypeGrid240 = 0
      TypeGrid120 = 0
      TypeGrid320 = 0
      TypeGrid160 = 0
      X = 2
      Y = 0
      Name
      IsMaster = False
      PowerSectorName
      Gaps:
        Left = 0
        Bottom = 0
        Right = 0
        Top = 0
        S4Left = 0
        S4Bottom = 0
        S4Right = 0
        S4Top = 0
      BorderID:
        Left = 0
        Bottom = 0
        Right = 0
        Top = 0
    Segment[10]:
      TypeGrid240 = 0
      TypeGrid120 = 0
      TypeGrid320 = 0
      TypeGrid160 = 0
      X = 2
      Y = 1
      Name
      IsMaster = False
      PowerSectorName
      Gaps:
        Left = 0
        Bottom = 0
        Right = 0
        Top = 0
        S4Left = 0
        S4Bottom = 0
        S4Right = 0
        S4Top = 0
      BorderID:
        Left = 0
        Bottom = 0
        Right = 0
        Top = 0
    Segment[11]:
      TypeGrid240 = 0
      TypeGrid120 = 0
      TypeGrid320 = 0
      TypeGrid160 = 0
      X = 2
      Y = 2
      Name
      IsMaster = False
      PowerSectorName
      Gaps:
        Left = 0
        Bottom = 0
        Right = 0
        Top = 0
        S4Left = 0
        S4Bottom = 0
        S4Right = 0
        S4Top = 0
      BorderID:
        Left = 0
        Bottom = 0
        Right = 0
        Top = 0
    Segment[12]:
      TypeGrid240 = 0
      TypeGrid120 = 0
      TypeGrid320 = 0
      TypeGrid160 = 0
      X = 2
      Y = 3
      Name
      IsMaster = False
      PowerSectorName
      Gaps:
        Left = 0
        Bottom = 0
        Right = 0
        Top = 0
        S4Left = 0
        S4Bottom = 0
        S4Right = 0
        S4Top = 0
      BorderID:
        Left = 0
        Bottom = 0
        Right = 0
        Top = 0
    Segment[13]:
      TypeGrid240 = 0
      TypeGrid120 = 0
      TypeGrid320 = 0
      TypeGrid160 = 0
      X = 3
      Y = 0
      Name
      IsMaster = False
      PowerSectorName
      Gaps:
        Left = 0
        Bottom = 0
        Right = 0
        Top = 0
        S4Left = 0
        S4Bottom = 0
        S4Right = 0
        S4Top = 0
      BorderID:
        Left = 0
        Bottom = 0
        Right = 0
        Top = 0
    Segment[14]:
      TypeGrid240 = 0
      TypeGrid120 = 0
      TypeGrid320 = 0
      TypeGrid160 = 0
      X = 3
      Y = 1
      Name
      IsMaster = False
      PowerSectorName
      Gaps:
        Left = 0
        Bottom = 0
        Right = 0
        Top = 0
        S4Left = 0
        S4Bottom = 0
        S4Right = 0
        S4Top = 0
      BorderID:
        Left = 0
        Bottom = 0
        Right = 0
        Top = 0
    Segment[15]:
      TypeGrid240 = 0
      TypeGrid120 = 0
      TypeGrid320 = 0
      TypeGrid160 = 0
      X = 3
      Y = 2
      Name
      IsMaster = False
      PowerSectorName
      Gaps:
        Left = 0
        Bottom = 0
        Right = 0
        Top = 0
        S4Left = 0
        S4Bottom = 0
        S4Right = 0
        S4Top = 0
      BorderID:
        Left = 0
        Bottom = 0
        Right = 0
        Top = 0
    Segment[16]:
      TypeGrid240 = 0
      TypeGrid120 = 0
      TypeGrid320 = 0
      TypeGrid160 = 0
      X = 3
      Y = 3
      Name
      IsMaster = False
      PowerSectorName
      Gaps:
        Left = 0
        Bottom = 0
        Right = 0
        Top = 0
        S4Left = 0
        S4Bottom = 0
        S4Right = 0
        S4Top = 0
      BorderID:
        Left = 0
        Bottom = 0
        Right = 0
        Top = 0
  Synchronization = NotUsed
```

### Config_2.assembly6d - X20EM0613/mapp6D/Config_2.assembly6d
```
Element gAssembly6D_1 (Type=assembly6d)
  Simulation6D = SimOff
  Ethernet6D:
    IpAddress = 192.168.125.239
    SubnetMask = 255.255.255.0
    Gateway = 192.168.125.1
  Shuttles:
    MaxShuttleCount = 8
    ShuttleIDMode = RealTimeID
    RealModeDetectionType = Any
    DefaultPosition:
      DefZ = 1.0
      DefRx = 0
      DefRy = 0
      DefRz = 0
    Limits:
      InPlaneLimits:
        InPlaneVelLim = 2
        InPlaneAccLim = 20
        InPlaneEmergDec = 20
      ShortAxLim:
        ShortAxAccLim:
          AccZLim = 10.0
          AccRxLim = 10.0
          AccRyLim = 10.0
          AccRzLim = 10.0
        ShortAxVelLim:
          VelZLim = 0.15
          VelRxLim = 0.1
          VelRyLim = 0.1
          VelRzLim = 0.3
  CyclicChannel6D:
    ReadChannel:
      Xaxis = TRUE
      Yaxis = TRUE
      Zaxis = TRUE
      Rxaxis = TRUE
      Ryaxis = TRUE
      Rzaxis = TRUE
  SystemReactions6D:
    LostCommReaction6D = Continue
  Fieldbus6D:
    SyncMode6D = ExternalPlkSync
    IFName = IF3
    NodeNumber = 239
  IOMapp:
    Input = ::gCommInput
    Output = ::gCommOutput
  Layout:
    Layout6D[1] = Layout6D_1
```

## Configuration Simulation

CPU X20EM0613, AutomationRuntime 6.0.2, Build 11.3.0, Vc 6.0.0

### Task classes (Cpu.sw)
```
Cyclic#1 (cycle 2000 us, tolerance 0 us):
  Acp6D <- Acp6D.Acp6D.prg
  Main <- Main.Main.prg
Cyclic#8:
  Robot <- Robot.Robot.prg
NcDataObjects: McDriveLog
Binaries: udbdef, mvLoader, mvConfig, OpcUaSrv, TCData, FWRules, ArSvcReg, BRRole, asfw, Role, ashwac, UaCsConfig, sysconf, iomap, Config_2, Config, Config_1, ashwd, User, arconfig
Libraries: runtime, AsIecCon, astime, operator, brfiDemo, RandLib, BrAbbRws, AsHttp, ArEventLog, Crypto, FileIO, AsBrStr, UaCoal, AsIODiag, standard, sys_lib, McAcp6DSys, UaCoalPrv, AsBrMath, ArSsl, strUtil, comUtil, AsTCP, brdkMU, MTFilter, AsUDP, MTLinAlg, MTTypes, brdkSTR, brsystem, AsSem, McAcp6D, McBase, MpBase
```

### Hardware
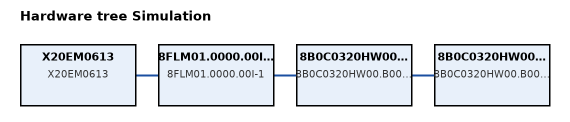
```
8B0C0320HW00.B00-1 : 8B0C0320HW00.B00-1 v1.0.1.3 (NodeNumber=3)  [PLK1 -> 8FLM01.0000.00I-1.PLK2 [Cable Type=PowerlinkCable, Length=10, Version=1.0.0.3]; PLK2 -> 8B0C0320HW00.B00-1_a.PLK1 [Cable Type=PowerlinkCable, Length=10, Version=1.0.0.3]]
  FunctionModel = DirectControl
  Supervision = off
  OutputVoltage = 58000
  CurrentLimitation = Used
  OutputCurrentLimit = 20000
  OutputCurrentLimitTime = 20
  ConfigOutputState = on
8B0C0320HW00.B00-1_a : 8B0C0320HW00.B00-1 v1.0.1.3  [PLK1 -> 8B0C0320HW00.B00-1.PLK2 [Cable Type=PowerlinkCable, Length=10, Version=1.0.0.3]]
  FunctionModel = DirectControl
  Supervision = off
  OutputVoltage = 58000
  CurrentLimitation = Used
  OutputCurrentLimit = 20000
  OutputCurrentLimitTime = 20
  ConfigOutputState = on
8FLM01.0000.00I-1 : 8FLM01.0000.00I-1 v1.0.0.1 (NodeNumber=239)  [PLK1 -> X20EM0613.IF3 [Cable Type=PowerlinkCable, Length=10, Version=1.0.0.3]; PLK2 -> 8B0C0320HW00.B00-1.PLK1 [Cable Type=PowerlinkCable, Length=10, Version=1.0.0.3]]
  Supervision = off
X20EM0613 : X20EM0613 v1.1.1.0
  Connector IF2:
    ActivateDevice = 1
    Mode = Manual
    InternetAddress = 192.168.125.201
    SubnetMask = 255.255.255.0
  ConfigurationID = Teknologia25_Config1
  Simulation = 1
  RemanentGlobalPvSize = 1024
  TimerDeviceType = EPLX2X
  TimerDevice = X20EM0613.IF3
  TaskClassIdleTime = 2000
  Cyclic1Duration = 2000
  Cyclic1Tolerance = 0
  Cyclic4Duration = 10000
  FileDevice1
  FileDeviceName1 = 6DData
  FileDevicePath1 = USER_PATH
  ActivateFtpServer = 1
  FTPProtocol = 1
  FtpUser1
  FtpUsername1 = br
  FtpUserPassword1 = QPRPBigPRs9A9gh3LdxcLXVCbSQ2d9xz/Uc992F9YlE=  // admin
  FtpUserSalt1 = 6+bIiqgw
  FTPAccessRight1 = 0
  FTPdevice1 = ALL
  ActivateWebServer = 1
  WebServerProtocol = 1
  WebServerPort = 8087
  ActivateSdm = 1
```

- Physical/Simulation/X20EM0613/IoMap.iom: same as Physical/Config1/X20EM0613/IoMap.iom
- Physical/Simulation/X20EM0613/mapp6D/Config_1.layout6d: same as Physical/Config1/X20EM0613/mapp6D/Config_1.layout6d
### Config_2.assembly6d - X20EM0613/mapp6D/Config_2.assembly6d
```
Element gAssembly6D_1 (Type=assembly6d)
  Simulation6D = SimOn
  Ethernet6D:
    IpAddress = 192.168.125.239
    SubnetMask = 255.255.255.0
    Gateway = 192.168.125.1
  Shuttles:
    MaxShuttleCount = 8
    ShuttleIDMode = RealTimeID
    RealModeDetectionType = Any
    DefaultPosition:
      DefZ = 1.0
      DefRx = 0
      DefRy = 0
      DefRz = 0
    Limits:
      InPlaneLimits:
        InPlaneVelLim = 2
        InPlaneAccLim = 20
        InPlaneEmergDec = 20
      ShortAxLim:
        ShortAxAccLim:
          AccZLim = 10.0
          AccRxLim = 10.0
          AccRyLim = 10.0
          AccRzLim = 10.0
        ShortAxVelLim:
          VelZLim = 0.15
          VelRxLim = 0.1
          VelRyLim = 0.1
          VelRzLim = 0.3
  CyclicChannel6D:
    ReadChannel:
      Xaxis = TRUE
      Yaxis = TRUE
      Zaxis = TRUE
      Rxaxis = TRUE
      Ryaxis = TRUE
      Rzaxis = TRUE
  SystemReactions6D:
    LostCommReaction6D = Continue
  Fieldbus6D:
    SyncMode6D = ExternalPlkSync
    IFName = IF3
    NodeNumber = 239
  IOMapp:
    Input = ::gCommInput
    Output = ::gCommOutput
  Layout:
    Layout6D[1] = Layout6D_1
```

## Logical view

Binary libraries used (declarations not repeated): operator, runtime, astime, AsIecCon, standard, AsBrStr, AsBrMath, FileIO, BrAbbRws 2.0.0, AsHttp, ArEventLog, ArSsl, Crypto 2.0.0, AsIODiag, AsSem, sys_lib, brsystem, MTFilter 6.0.0, MTTypes, MTLinAlg 6.0.0, AsUDP, AsTCP, McAcp6D 3.4.1, McBase, MpBase 6.0.0

### Global.typ - Global data types
```iecst
(*Main control datatype*)
(*Global shuttle array datatype*)

TYPE
	gShuttleListType : 	STRUCT  (*Global shuttle list datatype*)
		ID : UINT; (*ID of the shuttle*)
		Ref : Mc6DShuttleType; (*Reference to the shuttle*)
	END_STRUCT;
	gRobotTyp : 	STRUCT
		liftCup : BOOL;
		placeCup : BOOL;
		moveRobotHome : BOOL;
		AcoposWin : BOOL;
		CupCoordinate : gRobotParTyp;
		CupSelection : gRobotParTyp;
		Status : gRobotStatusTyp;
	END_STRUCT;
	gRobotParTyp : 	STRUCT
		X : REAL;
		Y : REAL;
	END_STRUCT;
	gRobotStatusTyp : 	STRUCT
		phaseOK : BOOL;
		phaseNum : REAL;
	END_STRUCT;
	gHMI_typ : 	STRUCT
		Precision : HMI_Precision_typ;
		Weight : HMI_Weight_typ;
		Stereotype : HMI_Stereotype_typ;
		Teach : HMI_Teach_typ;
		Zone : HMI_Zone_typ;
		ZoneDataProvider : ARRAY[0..49]OF STRING[40];
		ZoneDataIndex : USINT;
		ActivateZone : BOOL;
		shuttles : ARRAY[0..7]OF HMI_Shuttle_pos_typ;
		General : HMI_general_typ;
		Status : HMI_status_typ;
		Data : Motion6D_data_typ;
		Game : HMI_game_typ;
		Force : HMI_force_typ;
	END_STRUCT;
	HMI_Shuttle_pos_typ : 	STRUCT
		X : REAL;
		Y : REAL;
		RZ : REAL;
	END_STRUCT;
	HMI_Precision_typ : 	STRUCT
		Position : McAcp6DShPositionType;
		TargetPosition : McAcp6DShPositionType;
		Acceleration : REAL;
		Velocity : REAL;
	END_STRUCT;
	HMI_Teach_typ : 	STRUCT
		moveString : STRING[2000];
		update : BOOL;
	END_STRUCT;
	HMI_Weight_typ : 	STRUCT
		Position : McAcp6DShPositionType;
		Payload : REAL;
		StoreOffset : BOOL;
		NoMoveAllowed : BOOL;
	END_STRUCT;
	HMI_Stereotype_typ : 	STRUCT
		Size : McAcp6DPayloadSizeType;
	END_STRUCT;
	HMI_Zone_typ : 	STRUCT
		Active : HMI_zone_detail_typ;
		Preview : HMI_zone_detail_typ;
	END_STRUCT;
	HMI_zone_detail_typ : 	STRUCT
		BottomLeft : McAcp6DInPlaneAxesType;
		TopRight : McAcp6DInPlaneAxesType;
	END_STRUCT;
	gFeatureDemo_typ : 	STRUCT
		Active : BOOL;
		newZoneData : HMI_zone_detail_typ;
		newStereotypeData : McAcp6DPayloadSizeType;
		featureState : USINT;
		featureDemoState : USINT;
		returnState : USINT;
		zoneIndex : USINT;
		FB : gFeatureFB_typ;
		Cmd : gFeatureDemoCmds_typ;
		Int : gFeatureInternal_typ;
		Addition : gFeatureDemoAddition_typ;
	END_STRUCT;
	gFeatureDemoCmds_typ : 	STRUCT
		newZone : BOOL;
		newStereotype : BOOL;
		StopDemo : BOOL;
		StartDemo : BOOL;
	END_STRUCT;
	gFeatureFB_typ : 	STRUCT
		ZoneCreate : MC_BR_ZoneCreate_Acp6D;
		GetZone : MC_BR_AsmGetZone_Acp6D;
		ZoneOverride : MC_BR_ZoneOverride_Acp6D;
		StereoTypeDefine : MC_BR_ShStereotypeDefine_Acp6D;
		StereoTypeDelete : MC_BR_ShStereotypeDelete_Acp6D;
		GroupDelete : MC_BR_ShGroupDelete_Acp6D;
		GroupCreate : MC_BR_ShGroupCreate_Acp6D;
		GroupCoupleCtrl : MC_BR_ShGroupCoupleCtrl_Acp6D;
		GroupAddShuttle : MC_BR_ShGroupAddShuttle_Acp6D;
		R_TRIG_0 : R_TRIG;
		MoveInPlaneAsync : MC_BR_MoveInPlaneAsync_Acp6D;
		ReadInfo : ARRAY[0..7]OF MC_BR_ShReadInfo_Acp6D;
		StopAll : MC_BR_AsmStop_Acp6D;
		PowerOff : MC_BR_AsmPowerOff_Acp6D;
		PowerOn : MC_BR_AsmPowerOn_Acp6D;
		TON_1 : TON;
		TON_0 : TON;
		Reset : MC_BR_AsmReset_Acp6D;
	END_STRUCT;
	gFeatureInternal_typ : 	STRUCT
		ready : BOOL;
		z : USINT;
		i : USINT;
		tempSTR : STRING[20];
		tempSTR1 : STRING[20];
		zoneReset : BOOL;
		FirstRun : BOOL;
	END_STRUCT;
	HMI_general_typ : 	STRUCT
		PlayButton : BOOL;
		StopButton : BOOL;
		ResetButton : BOOL;
		BackToHome : BOOL;
		ResetPLC : BOOL;
	END_STRUCT;
	HMI_status_typ : 	STRUCT
		Running : USINT;
		ReadyToRun : USINT;
		Stopped : USINT;
		Error : USINT;
		AllowPlay : BOOL;
		AllowStop : BOOL;
		AllowReset : BOOL;
	END_STRUCT;
	HMI_game_typ : 	STRUCT
		Mode : USINT;
		Selection : USINT;
		CorrectShuttle : USINT;
		EndUserSelection : USINT;
		GameShuffleFinished : BOOL;
		GameFinished : BOOL;
		NewGame : BOOL;
		ExitGame : BOOL;
		GameRequested : BOOL;
		OpenGamePage : BOOL;
		GameState : USINT;
	END_STRUCT;
	gFeatureDemoAddition_typ : 	STRUCT
		Levitate : BOOL;
		Rotate : BOOL;
		Force : BOOL;
	END_STRUCT;
	HMI_force_typ : 	STRUCT
		mode : USINT;
		prevMode : USINT;
	END_STRUCT;
END_TYPE
```

### Global.var - Global variables
```iecst
(*Communication Variables*)
VAR
	gCommInput : Mc6DControllerFBIOType; (*Communication variable INPUT*)
	gCommOutput : Mc6DControllerFBIOType; (*Communication variable OUTPUT*)
END_VAR
(*Global Control Variable*)
VAR
	gShuttleList : ARRAY[0..gMAX_INDEX_SHUTTLE] OF gShuttleListType; (*Global shuttle list*)
	gShuttles : ARRAY[0..7] OF McAcp6DShPositionType;

	gHMI : gHMI_typ;
	gZones : ARRAY[0..49] OF HMI_Zone_typ;
	gFeatureDemo : gFeatureDemo_typ;
END_VAR
(**)
```

### Package Logical/Libraries - Global libraries

### Library Logical/Libraries/RandLib (ANSIC)

#### RandLib.fun - Exported functions and function blocks
```iecst
(********************************************************************
 * COPYRIGHT -- Bernecker + Rainer
 ********************************************************************
 * Library: RandLib
 * File: RandLib.fun
 * Author: manentiv
 * Created: December 20, 2011
 ********************************************************************
 * Functions and function blocks of library RandLib
 ********************************************************************)

FUNCTION RandValueDINT : DINT (*TODO: Add your comment here*)
	VAR_INPUT
		min : DINT;
		max : DINT;
	END_VAR
END_FUNCTION

FUNCTION RandValueREAL : REAL (*TODO: Add your comment here*)
	VAR_INPUT
		min : REAL;
		max : REAL;
	END_VAR
END_FUNCTION
```

#### RandValueREAL.c
```c
/********************************************************************
 * COPYRIGHT -- Bernecker + Rainer
 ********************************************************************
 * Library: RandLib
 * File: RandValue.c
 * Author: manentiv
 * Created: December 20, 2011
 ********************************************************************
 * Implementation of library RandLib
 ********************************************************************/

#include <bur/plctypes.h>
#ifdef __cplusplus
	extern "C"
	{
#endif

	#include "RandLib.h"
	#include <stdlib.h>
	#include <time.h>

#ifdef __cplusplus
	};
#endif

/* TODO: Add your comment here */
REAL RandValueREAL(REAL min, REAL max)
{
	REAL x;
	TIME t;
	t = clock_ms();
	/* Intializes random number generator */

	x = (float)(rand() % (int)max + (int)min);

	return x;
}
```

#### RandValueDINT.c
```c
/********************************************************************
 * COPYRIGHT -- Bernecker + Rainer
 ********************************************************************
 * Library: RandLib
 * File: RandValue.c
 * Author: manentiv
 * Created: December 20, 2011
 ********************************************************************
 * Implementation of library RandLib
 ********************************************************************/

#include <bur/plctypes.h>
#ifdef __cplusplus
	extern "C"
	{
#endif

	#include "RandLib.h"
	#include <stdlib.h>

#ifdef __cplusplus
	};
#endif

/* TODO: Add your comment here */
signed long RandValueDINT(signed long min, signed long max)
{
	DINT x;
	TIME t;
	t = clock_ms();
	/* Intializes random number generator */
	srand((unsigned) t);

	x = rand()%(max-min+1)+min;

	return x;
}
```

### Library Logical/Libraries/brdkMU (ANSIC, version 5.1.0) - BRDK machine unit library. Provides functionality to control machines.
Depends on: AsSem, sys_lib, brsystem, brdkSTR

- Library Logical/Libraries/brdkSTR (ANSIC, version 1.7.0) - brdk string handling library. Expands string functionality. (no source held here)

### Library Logical/Libraries/comUtil (ANSIC, version 1.0.4)
Depends on: AsTCP, standard, sys_lib, AsBrStr

#### comUtil.fun
```iecst
{REDUND_ERROR} FUNCTION_BLOCK ws_server (*TODO: Add your comment here*) (*$GROUP=User,$CAT=User,$GROUPICON=User.png,$CATICON=User.png*)
	VAR_INPUT
		Enable : BOOL;
		ServerPort : UINT;
	END_VAR
	VAR_OUTPUT
		Active : BOOL;
		httpPort : UDINT;
	END_VAR
	VAR
		Internal : ws_server_int_typ;
	END_VAR
END_FUNCTION_BLOCK

{REDUND_ERROR} FUNCTION pvValues : BOOL (*TODO: Add your comment here*) (*$GROUP=User,$CAT=User,$GROUPICON=User.png,$CATICON=User.png*)
	VAR_INPUT
		pPvName : UDINT;
		pBuffer : UDINT;
		BufferLen : UDINT;
	END_VAR
END_FUNCTION

{REDUND_ERROR} FUNCTION pvElements : BOOL (*TODO: Add your comment here*) (*$GROUP=User,$CAT=User,$GROUPICON=User.png,$CATICON=User.png*)
	VAR_INPUT
		pPvName : UDINT;
		pBuffer : UDINT;
		pParent : UDINT;
		last : BOOL;
		first : BOOL;
	END_VAR
END_FUNCTION

{REDUND_ERROR} FUNCTION_BLOCK PLC_var_info (*TODO: Add your comment here*) (*$GROUP=User,$CAT=User,$GROUPICON=User.png,$CATICON=User.png*)
	VAR_INPUT
		enable : BOOL;
	END_VAR
	VAR_OUTPUT
		active : BOOL;
	END_VAR
	VAR
		Internal : plc_var_info_typ;
	END_VAR
	VAR_INPUT
		browse : BOOL;
	END_VAR
	VAR_OUTPUT
		done : BOOL;
		data : Plc_typ;
	END_VAR
END_FUNCTION_BLOCK
```

#### Types.typ
```iecst
TYPE
	monitor_var_typ : 	STRUCT
		variables : ARRAY[0..MAX_MONITOR_VAR_MINUS1]OF var_typ;
		count : USINT;
		active : BOOL;
		init : BOOL;
	END_STRUCT;
	var_typ : 	STRUCT
		name : STRING[80];
		queryName : STRING[80];
		crc : UDINT;
		pv_addr : UDINT;
		datatype : UINT;
		size : UDINT;
		clientIdent : UDINT;
	END_STRUCT;
	ws_server_clients_typ : 	STRUCT
		client : ARRAY[0..MAX_CLIENT_COUNT_MINUS1]OF ws_server_client_typ;
		count : USINT;
	END_STRUCT;
	ws_server_client_data_typ : 	STRUCT
		recvbuf : ARRAY[0..9999]OF USINT;
		sendbuf : ARRAY[0..99999]OF USINT;
		recvlen : UDINT;
	END_STRUCT;
	ws_server_client_fb_typ : 	STRUCT
		TcpSend_0 : TcpSend;
		TcpRecv_0 : TcpRecv;
		TcpClose_0 : TcpClose;
		TON_0 : TON;
	END_STRUCT;
	ws_server_client_typ : 	STRUCT
		FB : ws_server_client_fb_typ;
		data : ws_server_client_data_typ;
		monitor : monitor_var_typ;
		ip_addr : STRING[20];
		commState : USINT;
		status : INT;
		ident : UDINT;
		monitorActive : BOOL;
	END_STRUCT;
	ws_server_data_typ : 	STRUCT
		ip_addr : STRING[20];
		monitorData : ARRAY[0..99999]OF USINT;
		latestData1 : ARRAY[0..99999]OF USINT;
		latestData : ARRAY[0..99999]OF USINT;
		prevError : UDINT;
	END_STRUCT;
	ws_server_fb_typ : 	STRUCT
		TcpOpen_0 : TcpOpen;
		TcpServer_0 : TcpServer;
		TcpClose_0 : TcpClose;
		TON_0 : TON;
		TcpIoctl_0 : TcpIoctl;
		PLC_var_info_0 : PLC_var_info;
	END_STRUCT;
	ws_server_int_typ : 	STRUCT
		FB : ws_server_fb_typ;
		data : ws_server_data_typ;
		clients : ws_server_clients_typ;
		read : monitor_var_typ;
		serverState : USINT;
	END_STRUCT;
	plc_var_info_typ : 	STRUCT
		plc : Plc_typ;
		var_typ : PV_xList_typ;
		module_typ : MO_List_typ;
		MO_info_0 : MO_info;
		browse_module_state : USINT;
		browse_var_state : USINT;
		prev_index : UINT;
		datatype : UDINT;
		datalen : UDINT;
		datadim : UINT;
		browse : BOOL;
		status : UINT;
		index : UINT;
		found : BOOL;
		localVarFound : BOOL;
		i : UINT;
		j : UINT;
		tempSTRING : STRING[80];
	END_STRUCT;
	Task_typ : 	STRUCT
		Name : STRING[20];
		StartAddress : UDINT;
		Size : UDINT;
		Version : ARRAY[0..9]OF USINT;
		Date : RTCtime_typ;
		Variables : ARRAY[0..200]OF Variable_typ;
		VariableCount : UINT;
	END_STRUCT;
	Plc_typ : 	STRUCT
		TaskCount : UINT;
		Tasks : ARRAY[0..20]OF Task_typ;
		GlobalVars : ARRAY[0..100]OF Variable_typ;
		GlobalVarCount : UINT;
	END_STRUCT;
	Variable_typ : 	STRUCT
		Name : STRING[32];
		Type : UINT;
	END_STRUCT;
END_TYPE
```
